TYPE AdasStreamSetup :
STRUCT
	blockType: USINT := 15;
	blockLength: USINT := 8;
	fillByte1: USINT;
	fillByte2: USINT;
	selectTrack: USINT;
	selectAxis: USINT;
	selectSignal: USINT;
	selectFlag: SINT;
END_STRUCT
END_TYPE

(* stored: Version 1.1.0.1, ProductVersion 3.1.4022.16
   DUT AdasStreamSetup: Id {301c71d5-a9d8-4b97-baf3-8ab88b15e5c0} *)
